(*
Allows registration of FB implementing `I_Execute`. 
*)
FUNCTION_BLOCK FINAL Execute IMPLEMENTS I_ExecuteNode, I_Debug
VAR
	_iExecute		: I_Execute;
	_iNext			: I_ExecuteNode;
	_nState			: Result;
	_nPhase			: INT;
END_VAR

METHOD INTERNAL Attach : Result
VAR_INPUT
	iExecute		: I_ExecuteNode;
END_VAR
VAR
	_iThis			: I_ExecuteNode := THIS^;
END_VAR
IF iExecute = 0 THEN
	DebugMsg(0, Tc2_Standard.CONCAT(__POUNAME(), ': Itf = 0!'));
	RETURN;
END_IF

IF _iThis <> _Runtime.iLastCyclic THEN
	DebugMsg(THIS^, Tc2_Standard.CONCAT(__POUNAME(), ': Is not the last node!'));
	RETURN;
END_IF

IF IsSome(iExecute.state) THEN
	DebugMsg(iExecute, Tc2_Standard.CONCAT(__POUNAME(), ': Has already been added!'));
	RETURN;
END_IF

_Runtime.iLastCyclic := iExecute;
_iNext := iExecute;
END_METHOD

METHOD INTERNAL Exe
VAR_OUTPUT
	iNext: I_ExecuteNode;
END_VAR
_iExecute.Execute(_nPhase);
iNext := _iNext;
END_METHOD

//FB_Init is always available implicitly and it is used primarily for initialization.
//The return value is not evaluated. For a specific influence, you can also declare the
//methods explicitly and provide additional code there with the standard initialization
//code. You can evaluate the return value.
{attribute 'hide'}
METHOD FB_Init: BOOL
VAR_INPUT
    bInitRetains: BOOL; // TRUE: the retain variables are initialized (reset warm / reset cold)
    bInCopyCode: BOOL;  // TRUE: the instance will be copied to the copy code afterward (online change)
	
	iExecute			: I_Execute;
END_VAR
IF IsSome(_nState) THEN
	RETURN;
END_IF

IF (_iExecute := iExecute) = 0 THEN
	_nState := Err.Itf0;
	DebugMsg(THIS^, Tc2_Standard.CONCAT(__POUNAME(), ': Itf = 0!'));
	RETURN;
END_IF



IF _Runtime.iLastCyclic <> 0 THEN
	IF IsErr(_Runtime.iLastCyclic.Attach(THIS^), nOut => _nState) THEN
		DebugMsg(THIS^, Tc2_Standard.CONCAT(__POUNAME(), ': Error Inside!'));
	END_IF
ELSE
	_Runtime.iFirstCyclic := THIS^;
	_Runtime.iLastCyclic := THIS^;
	_nState := Ok;
END_IF
END_METHOD

PROPERTY Phase : INT
GET
Phase := _nPhase;
END_GET
SET
_nPhase := Phase;
END_SET
END_PROPERTY

PROPERTY INTERNAL State : Result
GET
State := _nState;
END_GET
SET
IF IsNone(_nState) THEN
	_nState := State;
END_IF
END_SET
END_PROPERTY

END_FUNCTION_BLOCK

(* stored: Version 1.1.0.1
   POU Execute: Id {fd30bbbf-c4e7-4255-aff2-259a2cee51d5}, SpecialFunc None
   Method Attach: Id {aef47a4c-4a3d-4182-85d5-570cee5368fe}
   Method Exe: Id {c801d5e7-2cd0-4874-a9b5-b0187da63b5c}
   Method FB_init: Id {0c4d921f-e0eb-4cc3-851c-9a1e40abf9a1}
   Property Phase: Id {3dbfac59-95aa-4942-90ae-6bed7167a965}
   Get Get: Id {ee046bff-0af1-478c-bfb8-ca19ceb398e9}
   Set Set: Id {893ba47b-0fa2-41e5-bb90-b0e5e1297555}
   Property State: Id {24ee4fd7-b9b8-4900-937c-af456b6522b2}
   Get Get: Id {c6d174a2-5343-443e-acc0-fa6de12655a3}
   Set Set: Id {cdaef5bc-3e80-45aa-8a2d-58cc8bd11cfe} *)
